{attribute 'linkalways'} 
{attribute 'no_explicit_call' := 'This FB is a CLASS and must be accessed using methods or properties'}
{attribute 'enable_dynamic_creation'}
FUNCTION_BLOCK FINAL ABS_DWORD EXTENDS Node
VAR
	in : _DWORD(0);
	out : _DWORD(0);
END_VAR

METHOD PUBLIC Clone : I_Node
VAR
	pNode : POINTER TO ABS_DWORD;
END_VAR
pNode := __NEW(ABS_DWORD);
Clone := pNode^;
END_METHOD

METHOD FB_init : BOOL
VAR_INPUT
	bInitRetains : BOOL; // if TRUE, the retain variables are initialized (warm start / cold start)
	bInCopyCode : BOOL;  // if TRUE, the instance afterwards gets moved into the copy code (online change)
END_VAR
AddInput('in',THIS^.in);
AddOutput('out', THIS^.out);
END_METHOD

METHOD PROTECTED OnExecute
VAR
END_VAR
out.Value := ABS(in.Value);
END_METHOD

END_FUNCTION_BLOCK

(* stored: Version 1.1.0.1, ProductVersion 3.1.4024.15
   POU ABS_DWORD: Id {96a3fd51-06bb-4242-8563-55ca1872b9d5}, SpecialFunc None
   Folder Constructor: Id {aacd4f54-0311-4f23-89ea-3a354b69621f}
   Method Clone: Id {e72c4712-4779-4ad5-93f1-9d8572a24ecb}
   Method FB_init: Id {20fef6c1-c376-406c-85ff-ca426342ac11}
   Method OnExecute: Id {131393f4-625f-4ca5-a190-941e85f5e7f2} *)
